TYPE ST_ACswitchgear_set :
STRUCT
	b_inputContactorClose 	: BOOL;
	b_inputContactorOpen	: BOOL;
	b_EnableSynchronizer	: BOOL;
END_STRUCT
END_TYPE

(* stored: Version 1.1.0.1, ProductVersion 3.1.4026.18
   DUT ST_ACswitchgear_set: Id {2f66a9af-8538-48aa-a736-b263649b5802} *)
